(* PLC project PLC, Beckhoff Automation GmbH TwinCAT PLC Control 3.5.21.60 *)
(* stored: creationDateTime 2026-08-05T00:24:44.8344467, modificationDateTime 2026-08-05T00:24:44.8354582 *)

FUNCTION_BLOCK FB_SerialCom
VAR_IN_OUT
	bSendString		:BOOL;
	bClear			:BOOL;
END_VAR
VAR_INPUT
	sSendString		:STRING;
	sSuffix			:STRING := '$R$N';
END_VAR
VAR_OUTPUT
	sLastReceivedString	: STRING;
	bStringReceived		: BOOL;
	bReceiveBusy		: BOOL;
	bReceiveError		: BOOL;
	eReceiveErrorID		: ComError_t;
END_VAR
VAR
	RxBufferEL			: ComBuffer;	(* Receive data buffer; used with all receive function blocks *)
	TxBufferEL			: ComBuffer;	(* Transmit data buffer; used with all receive function blocks *)

	(* background communication with the EL6001 terminal *)
	fbEL6001Ctrl		: SerialLineControl;
	bEL6001CtrlError	: BOOL;
	eEL6001CtrlErrorID	: ComError_t;
	(* 	I/O variables for a EL6001 terminal*)
	stIn_EL6001 AT %I*	: EL6inData22B;	(* linked to the EL6001 in the TwinCAT System Manager *)
	stOut_EL6001 AT %Q*	: EL6outData22B;(* linked to the EL6001 in the TwinCAT System Manager *)

	Timer				: TON := (PT:=T#1S);
	fbSend				: SendString;
	bSendBusy			: BOOL;
	eSendErrorID		: ComError_t;

	fbReceive			: ReceiveString;
	sReceivedString		: STRING;
	bReceiveTimeout		: BOOL;
	nReceiveCounter		: UDINT;

	nSuffixPosition		: INT;
	ClearBuffer			: ClearComBuffer;
	
END_VAR

            (* background communication with the EL6001 terminal *)
fbEL6001Ctrl(
	Mode:= SERIALLINEMODE_EL6_22B, 
	pComIn:= ADR(stIn_EL6001), 
	pComOut:= ADR(stOut_EL6001), 
	SizeComIn:= SIZEOF(stIn_EL6001), 
	Error=> , 
	ErrorID=> , 
	TxBuffer:= TxBufferEL, 
	RxBuffer:= RxBufferEL );
IF fbEL6001Ctrl.Error THEN
	bEL6001CtrlError := TRUE;
	eEL6001CtrlErrorID := fbEL6001Ctrl.ErrorID;
END_IF

IF bSendString THEN
	fbSend(
		SendString:= CONCAT(sSendString, sSuffix),
		TXbuffer:= TxBufferEL,
		Busy=> bSendBusy,
		Error=> );
	sLastReceivedString := '';
	bSendString := FALSE;
END_IF

IF fbSend.Error <> COMERROR_NOERROR THEN
	eSendErrorID := fbSend.Error;
END_IF			
			
//	Receive string data:
fbReceive(
	Prefix:= ,
	Suffix:= sSuffix,
	Timeout:= T#1s,
	ReceivedString:= sReceivedString,
	RXbuffer:= RxBufferEL,
	StringReceived=> bStringReceived,
	Busy=> bReceiveBusy,
	Error=> ,
	RxTimeout=> bReceiveTimeout );
	
IF fbReceive.Error <> COMERROR_NOERROR THEN
	eReceiveErrorID := fbReceive.Error;
END_IF
IF bStringReceived THEN
	nReceiveCounter := nReceiveCounter + 1;
	nSuffixPosition := FIND (sReceivedString, sSuffix);
	sLastReceivedString := DELETE(sReceivedString,2,nSuffixPosition);
END_IF

IF bClear THEN
	ClearBuffer(Buffer := RxBufferEL);
	ClearBuffer(Buffer := TxBufferEL);
	bClear := FALSE;
END_IF


          
END_FUNCTION_BLOCK
